{region '#Template'}
	{attribute 'Version' := '5.1.0.0'}
	{attribute 'Tags' := '"LCID": "1031", "Text": "Gebäudeautomation, Kommunikation, Server, Client, Publisher, Subscriber"'}
	{attribute 'Tags' := '"LCID": "1033", "Text": "Building automation, Communication, Server, Client, Publisher, Subscriber"'}
	{attribute 'Using' := '"Type": "Template", "URI": "Site"'}
	{attribute 'Description' := '"LCID": "1031", "Text": "Server Datenkommunikation"'}
	{attribute 'Description' := '"LCID": "1033", "Text": "Server data communication"'}
{endregion}

FUNCTION_BLOCK FB_BA_AdsComServer_DGWS
VAR_INPUT CONSTANT
	BuildingSunBlind		: FB_BA_RawPublisher;
	arrFacadeData			: ARRAY[1..BA2_Param.nMaxNumberOfFacades] OF FB_BA_RawPublisher;
END_VAR

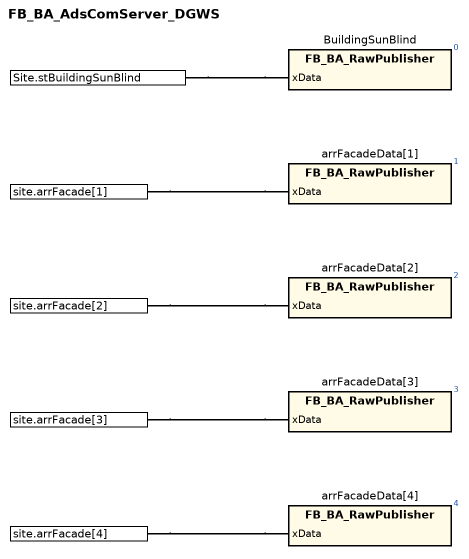
BuildingSunBlind(xData := Site.stBuildingSunBlind); // FB_BA_RawPublisher
arrFacadeData[1](xData := site.arrFacade[1]); // FB_BA_RawPublisher
arrFacadeData[2](xData := site.arrFacade[2]); // FB_BA_RawPublisher
arrFacadeData[3](xData := site.arrFacade[3]); // FB_BA_RawPublisher
arrFacadeData[4](xData := site.arrFacade[4]); // FB_BA_RawPublisher

END_FUNCTION_BLOCK

(* stored: Version 1.1.0.1, ProductVersion 3.1.4024.12
   POU FB_BA_AdsComServer_DGWS: Id {f1cf2108-6b12-48ae-ae74-1c680392c3da}, SpecialFunc None *)
